Omron Sysmac Studio project INV00x_MX2_ECT (Sysmac Studio 1.45.1.64010, LibraryProject)
(* Functionblocks that can be used for controlling 3G3MX2 with Omron NJ controller over EtherCAT communication. *)

# Controller new_Controller_0: NX102-9000 version 1.40
Task PrimaryTask (priority 4, period or condition 1000): DEMO_INV012_MX2_Analog_inputs, DEMO_INV000_MX2_Alarm, DEMO_INV001_MX2_ECT, DEMO_INV002_MX2_ECT, DEMO_INV003_MX2_ECT, DEMO_INV010_MX2_ExternalTrip, DEMO_INV011_MX2_Intelligent_inputs

TYPE INV00x_MX2\uWORD_BOOL_MX2 : UNION
    bit : ARRAY[0..15] OF BOOL;
    ch : WORD;
END_UNION END_TYPE
TYPE INV00x_MX2\uBYTE_BOOL_MX2 : UNION
    bit : ARRAY[0..7] OF BOOL;
    value : BYTE;
END_UNION END_TYPE

PROGRAM DEMO_INV000_MX2_Alarm
VAR
    sFB_Activate : BOOL;
    MX2 : INV001_MX2_ECT;
    sFrequence : REAL;
    sFwd : BOOL;
    sRev : BOOL;
    sFault_Reset : BOOL;
    sDuring_FDW : BOOL;
    sDuring_Rev : BOOL;
    sWarning : BOOL;
    sRemote : BOOL;
    sFreq_Match : BOOL;
    sConection_Error : BOOL;
    sFB_Activate_2 : BOOL;
    MX2_2 : INV002_MX2_ECT;
    sFault : BOOL;
    sFrequency_in : REAL;
    sFrequency_out : REAL;
    sFB_Activate_3 : BOOL;
    MX2_3 : INV003_MX2_ECT;
    sAcceleration : REAL;
    sDeceleration : REAL;
    MX2_Alarm : INV000_MX2_Alarm;
    sAlarm_Fault : STRING[256];
    sAlarm_Status : STRING[256];
    sAlarm_code : UINT;
    SDO_Obj_W : _sSDO_ACCESS;
END_VAR
VAR RETAIN
    Write_Data : WORD;
END_VAR
VAR
    EtherCAT_Write_External_Trip : EC_CoESDOWrite;
    Node : UINT;
    MX2_ExternalTrip : INV010_MX2_ExternalTrip;
    ExternalTrip : BOOL;
    Read_DI : BOOL;
    TEST : BOOL;
    test2 : WORD;
    s1 : BOOL;
    s2 : BOOL;
    s3 : BOOL;
    s4 : BOOL;
    s5 : BOOL;
    s6 : BOOL;
    s7 : BOOL;
    sRun_Command : BOOL;
    sRotation_Direction : BOOL;
    sExternal_Trip : BOOL;
    MX2_Intelligent_inputs : INV011_MX2_Intelligent_inputs;
    Analog_Input : BOOL;
    MX2_Analog_Inputs : INV012_MX2_Analog_inputs;
    sAnaloge_Value : REAL;
    MX2_Frequency_reference : UINT;
    MX2_Output_frequency_monitor : UINT;
    MX2_F002_1st_Acceleration_Time_1 : UDINT;
    MX2_F003_1st_Deceleration_Time_1 : UDINT;
    MX2_Coil_Data_0 : WORD;
    MX2_Command : WORD;
    MX2_d081_Fault_Monitor_1_Cause : UINT;
    MX2_d081_Fault_Monitor_1_Inverter_Status : UINT;
    MX2_d130_Analog_voltage_input_FV_monitor : UINT;
    MX2_Status : WORD;
END_VAR

(* Section Section1: ladder, written here as Structured Text *)

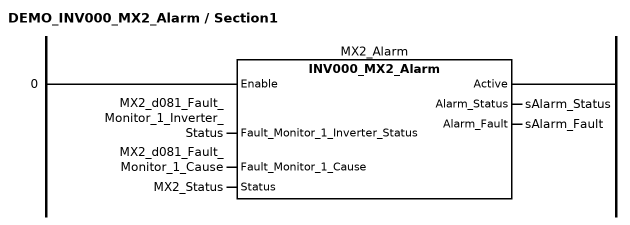
(* Rung 0 *)
MX2_Alarm(Enable := TRUE, Fault_Monitor_1_Inverter_Status := MX2_d081_Fault_Monitor_1_Inverter_Status, Fault_Monitor_1_Cause := MX2_d081_Fault_Monitor_1_Cause, Status := MX2_Status, Alarm_Status => sAlarm_Status, Alarm_Fault => sAlarm_Fault);
END_PROGRAM

PROGRAM DEMO_INV001_MX2_ECT
VAR
    sFB_Activate : BOOL;
    MX2 : INV001_MX2_ECT;
    sFrequence : REAL;
    sFwd : BOOL;
    sRev : BOOL;
    sFault_Reset : BOOL;
    sDuring_FDW : BOOL;
    sDuring_Rev : BOOL;
    sWarning : BOOL;
    sRemote : BOOL;
    sFreq_Match : BOOL;
    sConection_Error : BOOL;
    sFB_Activate_2 : BOOL;
    MX2_2 : INV002_MX2_ECT;
    sFault : BOOL;
    sFrequency_in : REAL;
    sFrequency_out : REAL;
    sFB_Activate_3 : BOOL;
    MX2_3 : INV003_MX2_ECT;
    sAcceleration : REAL;
    sDeceleration : REAL;
    MX2_Alarm : INV000_MX2_Alarm;
    sAlarm_Fault : STRING[256];
    sAlarm_Status : STRING[256];
    sAlarm_code : UINT;
    SDO_Obj_W : _sSDO_ACCESS;
END_VAR
VAR RETAIN
    Write_Data : WORD;
END_VAR
VAR
    EtherCAT_Write_External_Trip : EC_CoESDOWrite;
    Node : UINT;
    MX2_ExternalTrip : INV010_MX2_ExternalTrip;
    ExternalTrip : BOOL;
    Read_DI : BOOL;
    TEST : BOOL;
    test2 : WORD;
    s1 : BOOL;
    s2 : BOOL;
    s3 : BOOL;
    s4 : BOOL;
    s5 : BOOL;
    s6 : BOOL;
    s7 : BOOL;
    sRun_Command : BOOL;
    sRotation_Direction : BOOL;
    sExternal_Trip : BOOL;
    MX2_Intelligent_inputs : INV011_MX2_Intelligent_inputs;
    Analog_Input : BOOL;
    MX2_Analog_Inputs : INV012_MX2_Analog_inputs;
    sAnaloge_Value : REAL;
    MX2_F002_1st_Acceleration_Time_1 : UDINT;
    MX2_F003_1st_Deceleration_Time_1 : UDINT;
    MX2_d081_Fault_Monitor_1_Inverter_Status : UINT;
    MX2_d081_Fault_Monitor_1_Cause : UINT;
    MX2_Coil_Data_0 : WORD;
    MX2_d130_Analog_voltage_input_FV_monitor : UINT;
    sFrequency_0Hz_Warning : BOOL;
    MX2_Frequency_reference : UINT;
    MX2_Output_frequency_monitor : UINT;
    MX2_Command : WORD;
    MX2_Status : WORD;
END_VAR

(* Section Section1: ladder, written here as Structured Text *)

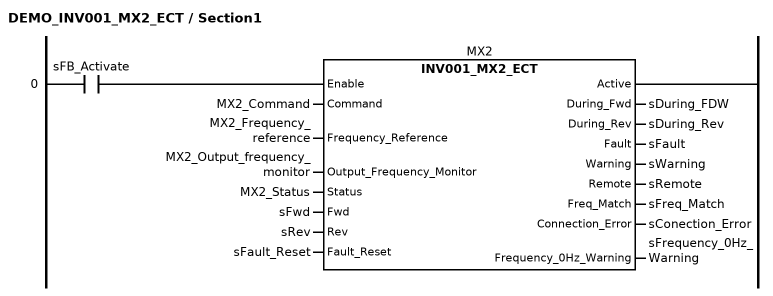
(* Rung 0 *)
MX2(Enable := sFB_Activate, Command := MX2_Command, Frequency_Reference := MX2_Frequency_reference, Output_Frequency_Monitor := MX2_Output_frequency_monitor, Status := MX2_Status, Fwd := sFwd, Rev := sRev, Fault_Reset := sFault_Reset, During_Fwd => sDuring_FDW, During_Rev => sDuring_Rev, Fault => sFault, Warning => sWarning, Remote => sRemote, Freq_Match => sFreq_Match, Connection_Error => sConection_Error, Frequency_0Hz_Warning => sFrequency_0Hz_Warning);
END_PROGRAM

PROGRAM DEMO_INV002_MX2_ECT
VAR
    sFB_Activate : BOOL;
    MX2 : INV001_MX2_ECT;
    sFrequence : REAL;
    sFwd : BOOL;
    sRev : BOOL;
    sFault_Reset : BOOL;
    sDuring_FDW : BOOL;
    sDuring_Rev : BOOL;
    sWarning : BOOL;
    sRemote : BOOL;
    sFreq_Match : BOOL;
    sConection_Error : BOOL;
    sFB_Activate_2 : BOOL;
    MX2_2 : INV002_MX2_ECT;
    sFault : BOOL;
    sFrequency_in : REAL;
    sFrequency_out : REAL;
    sFB_Activate_3 : BOOL;
    MX2_3 : INV003_MX2_ECT;
    sAcceleration : REAL;
    sDeceleration : REAL;
    MX2_Alarm : INV000_MX2_Alarm;
    sAlarm_Fault : STRING[256];
    sAlarm_Status : STRING[256];
    sAlarm_code : UINT;
    SDO_Obj_W : _sSDO_ACCESS;
END_VAR
VAR RETAIN
    Write_Data : WORD;
END_VAR
VAR
    EtherCAT_Write_External_Trip : EC_CoESDOWrite;
    Node : UINT;
    MX2_ExternalTrip : INV010_MX2_ExternalTrip;
    ExternalTrip : BOOL;
    Read_DI : BOOL;
    TEST : BOOL;
    test2 : WORD;
    s1 : BOOL;
    s2 : BOOL;
    s3 : BOOL;
    s4 : BOOL;
    s5 : BOOL;
    s6 : BOOL;
    s7 : BOOL;
    sRun_Command : BOOL;
    sRotation_Direction : BOOL;
    sExternal_Trip : BOOL;
    MX2_Intelligent_inputs : INV011_MX2_Intelligent_inputs;
    Analog_Input : BOOL;
    MX2_Analog_Inputs : INV012_MX2_Analog_inputs;
    sAnaloge_Value : REAL;
    MX2_Command : WORD;
    MX2_Frequency_reference : UINT;
    MX2_Output_frequency_monitor : UINT;
    MX2_Status : WORD;
    MX2_F002_1st_Acceleration_Time_1 : UDINT;
    MX2_F003_1st_Deceleration_Time_1 : UDINT;
    MX2_d081_Fault_Monitor_1_Inverter_Status : UINT;
    MX2_d081_Fault_Monitor_1_Cause : UINT;
    MX2_Coil_Data_0 : WORD;
    MX2_d130_Analog_voltage_input_FV_monitor : UINT;
    sFrequency_0Hz_Warning : BOOL;
END_VAR

(* Section Section1: ladder, written here as Structured Text *)

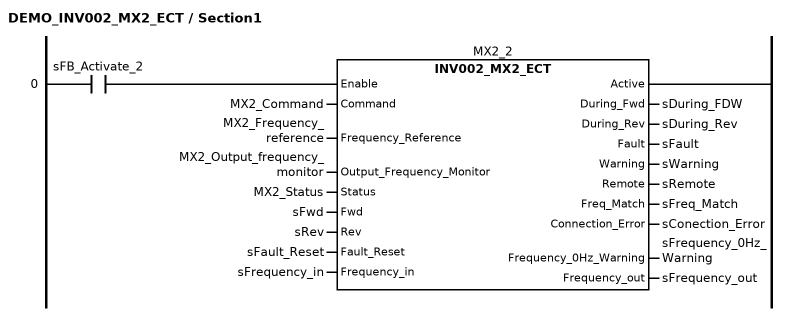
(* Rung 0 *)
MX2_2(Enable := sFB_Activate_2, Command := MX2_Command, Frequency_Reference := MX2_Frequency_reference, Output_Frequency_Monitor := MX2_Output_frequency_monitor, Status := MX2_Status, Fwd := sFwd, Rev := sRev, Fault_Reset := sFault_Reset, Frequency_in := sFrequency_in, During_Fwd => sDuring_FDW, During_Rev => sDuring_Rev, Fault => sFault, Warning => sWarning, Remote => sRemote, Freq_Match => sFreq_Match, Connection_Error => sConection_Error, Frequency_0Hz_Warning => sFrequency_0Hz_Warning, Frequency_out => sFrequency_out);
END_PROGRAM

PROGRAM DEMO_INV003_MX2_ECT
VAR
    sFB_Activate : BOOL;
    MX2 : INV001_MX2_ECT;
    sFrequence : REAL;
    sFwd : BOOL;
    sRev : BOOL;
    sFault_Reset : BOOL;
    sDuring_FDW : BOOL;
    sDuring_Rev : BOOL;
    sWarning : BOOL;
    sRemote : BOOL;
    sFreq_Match : BOOL;
    sConection_Error : BOOL;
    sFB_Activate_2 : BOOL;
    MX2_2 : INV002_MX2_ECT;
    sFault : BOOL;
    sFrequency_in : REAL;
    sFrequency_out : REAL;
    sFB_Activate_3 : BOOL;
    MX2_3 : INV003_MX2_ECT;
    sAcceleration : REAL;
    sDeceleration : REAL;
    MX2_Alarm : INV000_MX2_Alarm;
    sAlarm_Fault : STRING[256];
    sAlarm_Status : STRING[256];
    sAlarm_code : UINT;
    SDO_Obj_W : _sSDO_ACCESS;
END_VAR
VAR RETAIN
    Write_Data : WORD;
END_VAR
VAR
    EtherCAT_Write_External_Trip : EC_CoESDOWrite;
    Node : UINT;
    MX2_ExternalTrip : INV010_MX2_ExternalTrip;
    ExternalTrip : BOOL;
    Read_DI : BOOL;
    TEST : BOOL;
    test2 : WORD;
    s1 : BOOL;
    s2 : BOOL;
    s3 : BOOL;
    s4 : BOOL;
    s5 : BOOL;
    s6 : BOOL;
    s7 : BOOL;
    sRun_Command : BOOL;
    sRotation_Direction : BOOL;
    sExternal_Trip : BOOL;
    MX2_Intelligent_inputs : INV011_MX2_Intelligent_inputs;
    Analog_Input : BOOL;
    MX2_Analog_Inputs : INV012_MX2_Analog_inputs;
    sAnaloge_Value : REAL;
    MX2_Command : WORD;
    MX2_Frequency_reference : UINT;
    MX2_Output_frequency_monitor : UINT;
    MX2_Status : WORD;
    MX2_F002_1st_Acceleration_Time_1 : UDINT;
    MX2_F003_1st_Deceleration_Time_1 : UDINT;
    MX2_d081_Fault_Monitor_1_Inverter_Status : UINT;
    MX2_d081_Fault_Monitor_1_Cause : UINT;
    MX2_Coil_Data_0 : WORD;
    MX2_d130_Analog_voltage_input_FV_monitor : UINT;
    sFrequency_0Hz_Warning : BOOL;
END_VAR

(* Section Section1: ladder, written here as Structured Text *)

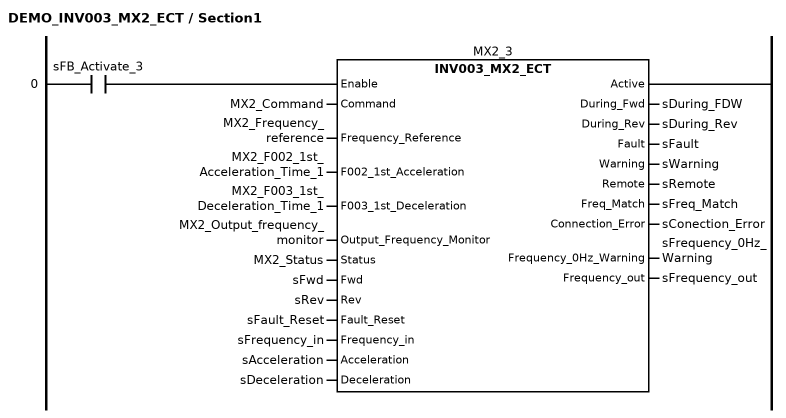
(* Rung 0 *)
MX2_3(Enable := sFB_Activate_3, Command := MX2_Command, Frequency_Reference := MX2_Frequency_reference, F002_1st_Acceleration := MX2_F002_1st_Acceleration_Time_1, F003_1st_Deceleration := MX2_F003_1st_Deceleration_Time_1, Output_Frequency_Monitor := MX2_Output_frequency_monitor, Status := MX2_Status, Fwd := sFwd, Rev := sRev, Fault_Reset := sFault_Reset, Frequency_in := sFrequency_in, Acceleration := sAcceleration, Deceleration := sDeceleration, During_Fwd => sDuring_FDW, During_Rev => sDuring_Rev, Fault => sFault, Warning => sWarning, Remote => sRemote, Freq_Match => sFreq_Match, Connection_Error => sConection_Error, Frequency_0Hz_Warning => sFrequency_0Hz_Warning, Frequency_out => sFrequency_out);
END_PROGRAM

PROGRAM DEMO_INV010_MX2_ExternalTrip
VAR
    sFB_Activate : BOOL;
    MX2 : INV001_MX2_ECT;
    sFrequence : REAL;
    sFwd : BOOL;
    sRev : BOOL;
    sFault_Reset : BOOL;
    sDuring_FDW : BOOL;
    sDuring_Rev : BOOL;
    sWarning : BOOL;
    sRemote : BOOL;
    sFreq_Match : BOOL;
    sConection_Error : BOOL;
    sFB_Activate_2 : BOOL;
    MX2_2 : INV002_MX2_ECT;
    sFault : BOOL;
    sFrequency_in : REAL;
    sFrequency_out : REAL;
    sFB_Activate_3 : BOOL;
    MX2_3 : INV003_MX2_ECT;
    sAcceleration : REAL;
    sDeceleration : REAL;
    MX2_Alarm : INV000_MX2_Alarm;
    sAlarm_Fault : STRING[256];
    sAlarm_Status : STRING[256];
    sAlarm_code : UINT;
    SDO_Obj_W : _sSDO_ACCESS;
END_VAR
VAR RETAIN
    Write_Data : WORD;
END_VAR
VAR
    EtherCAT_Write_External_Trip : EC_CoESDOWrite;
    Node : UINT;
    MX2_ExternalTrip : INV010_MX2_ExternalTrip;
    ExternalTrip : BOOL;
    Read_DI : BOOL;
    TEST : BOOL;
    test2 : WORD;
    s1 : BOOL;
    s2 : BOOL;
    s3 : BOOL;
    s4 : BOOL;
    s5 : BOOL;
    s6 : BOOL;
    s7 : BOOL;
    sRun_Command : BOOL;
    sRotation_Direction : BOOL;
    sExternal_Trip : BOOL;
    MX2_Intelligent_inputs : INV011_MX2_Intelligent_inputs;
    Analog_Input : BOOL;
    MX2_Analog_Inputs : INV012_MX2_Analog_inputs;
    sAnaloge_Value : REAL;
    MX2_Command : WORD;
    MX2_Frequency_reference : UINT;
    MX2_Output_frequency_monitor : UINT;
    MX2_Status : WORD;
    MX2_F002_1st_Acceleration_Time_1 : UDINT;
    MX2_F003_1st_Deceleration_Time_1 : UDINT;
    MX2_d081_Fault_Monitor_1_Inverter_Status : UINT;
    MX2_d081_Fault_Monitor_1_Cause : UINT;
    MX2_Coil_Data_0 : WORD;
    MX2_d130_Analog_voltage_input_FV_monitor : UINT;
END_VAR

(* Section Section1: ladder, written here as Structured Text *)

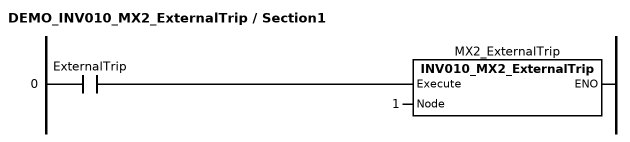
(* Rung 0 *)
MX2_ExternalTrip(Execute := ExternalTrip, Node := 1);
END_PROGRAM

PROGRAM DEMO_INV011_MX2_Intelligent_inputs
VAR
    sFB_Activate : BOOL;
    MX2 : INV001_MX2_ECT;
    sFrequence : REAL;
    sFwd : BOOL;
    sRev : BOOL;
    sFault_Reset : BOOL;
    sDuring_FDW : BOOL;
    sDuring_Rev : BOOL;
    sWarning : BOOL;
    sRemote : BOOL;
    sFreq_Match : BOOL;
    sConection_Error : BOOL;
    sFB_Activate_2 : BOOL;
    MX2_2 : INV002_MX2_ECT;
    sFault : BOOL;
    sFrequency_in : REAL;
    sFrequency_out : REAL;
    sFB_Activate_3 : BOOL;
    MX2_3 : INV003_MX2_ECT;
    sAcceleration : REAL;
    sDeceleration : REAL;
    MX2_Alarm : INV000_MX2_Alarm;
    sAlarm_Fault : STRING[256];
    sAlarm_Status : STRING[256];
    sAlarm_code : UINT;
    SDO_Obj_W : _sSDO_ACCESS;
END_VAR
VAR RETAIN
    Write_Data : WORD;
END_VAR
VAR
    EtherCAT_Write_External_Trip : EC_CoESDOWrite;
    Node : UINT;
    MX2_ExternalTrip : INV010_MX2_ExternalTrip;
    ExternalTrip : BOOL;
    Read_DI : BOOL;
    TEST : BOOL;
    test2 : WORD;
    s1 : BOOL;
    s2 : BOOL;
    s3 : BOOL;
    s4 : BOOL;
    s5 : BOOL;
    s6 : BOOL;
    s7 : BOOL;
    sRun_Command : BOOL;
    sRotation_Direction : BOOL;
    sExternal_Trip : BOOL;
    MX2_Intelligent_inputs : INV011_MX2_Intelligent_inputs;
    Analog_Input : BOOL;
    MX2_Analog_Inputs : INV012_MX2_Analog_inputs;
    sAnaloge_Value : REAL;
    MX2_Command : WORD;
    MX2_Frequency_reference : UINT;
    MX2_Output_frequency_monitor : UINT;
    MX2_Status : WORD;
    MX2_F002_1st_Acceleration_Time_1 : UDINT;
    MX2_F003_1st_Deceleration_Time_1 : UDINT;
    MX2_d081_Fault_Monitor_1_Inverter_Status : UINT;
    MX2_d081_Fault_Monitor_1_Cause : UINT;
    MX2_Coil_Data_0 : WORD;
    MX2_d130_Analog_voltage_input_FV_monitor : UINT;
END_VAR

(* Section Section1: ladder, written here as Structured Text *)

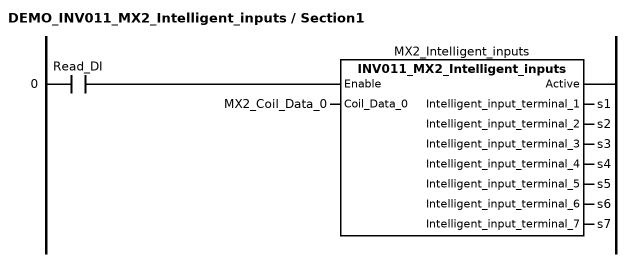
(* Rung 0 *)
MX2_Intelligent_inputs(Enable := Read_DI, Coil_Data_0 := MX2_Coil_Data_0, Intelligent_input_terminal_1 => s1, Intelligent_input_terminal_2 => s2, Intelligent_input_terminal_3 => s3, Intelligent_input_terminal_4 => s4, Intelligent_input_terminal_5 => s5, Intelligent_input_terminal_6 => s6, Intelligent_input_terminal_7 => s7);
END_PROGRAM

PROGRAM DEMO_INV012_MX2_Analog_inputs
VAR
    sFB_Activate : BOOL;
    MX2 : INV001_MX2_ECT;
    sFrequence : REAL;
    sFwd : BOOL;
    sRev : BOOL;
    sFault_Reset : BOOL;
    sDuring_FDW : BOOL;
    sDuring_Rev : BOOL;
    sWarning : BOOL;
    sRemote : BOOL;
    sFreq_Match : BOOL;
    sConection_Error : BOOL;
    sFB_Activate_2 : BOOL;
    MX2_2 : INV002_MX2_ECT;
    sFault : BOOL;
    sFrequency_in : REAL;
    sFrequency_out : REAL;
    sFB_Activate_3 : BOOL;
    MX2_3 : INV003_MX2_ECT;
    sAcceleration : REAL;
    sDeceleration : REAL;
    MX2_Alarm : INV000_MX2_Alarm;
    sAlarm_Fault : STRING[256];
    sAlarm_Status : STRING[256];
    sAlarm_code : UINT;
    SDO_Obj_W : _sSDO_ACCESS;
END_VAR
VAR RETAIN
    Write_Data : WORD;
END_VAR
VAR
    EtherCAT_Write_External_Trip : EC_CoESDOWrite;
    Node : UINT;
    MX2_ExternalTrip : INV010_MX2_ExternalTrip;
    ExternalTrip : BOOL;
    Read_DI : BOOL;
    TEST : BOOL;
    test2 : WORD;
    s1 : BOOL;
    s2 : BOOL;
    s3 : BOOL;
    s4 : BOOL;
    s5 : BOOL;
    s6 : BOOL;
    s7 : BOOL;
    sRun_Command : BOOL;
    sRotation_Direction : BOOL;
    sExternal_Trip : BOOL;
    MX2_Intelligent_inputs : INV011_MX2_Intelligent_inputs;
    Analog_Input : BOOL;
    MX2_Analog_Inputs : INV012_MX2_Analog_inputs;
    sAnaloge_voltage : REAL;
    sAnaloge_current : REAL;
    sAnaloge_voltage_Procentage : REAL;
    sAnaloge_current_Procentage : REAL;
    sAnaloge_voltage_Percentage : REAL;
    sAnaloge_current_Percentage : REAL;
    MX2_Command : WORD;
    MX2_Frequency_reference : UINT;
    MX2_Output_frequency_monitor : UINT;
    MX2_Status : WORD;
    MX2_F002_1st_Acceleration_Time_1 : UDINT;
    MX2_F003_1st_Deceleration_Time_1 : UDINT;
    MX2_d081_Fault_Monitor_1_Inverter_Status : UINT;
    MX2_d081_Fault_Monitor_1_Cause : UINT;
    MX2_Coil_Data_0 : WORD;
    MX2_d130_Analog_voltage_input_FV_monitor : UINT;
    MX2_d131_Analog_current_input_FI_monitor : UINT;
END_VAR

(* Section Section1: ladder, written here as Structured Text *)

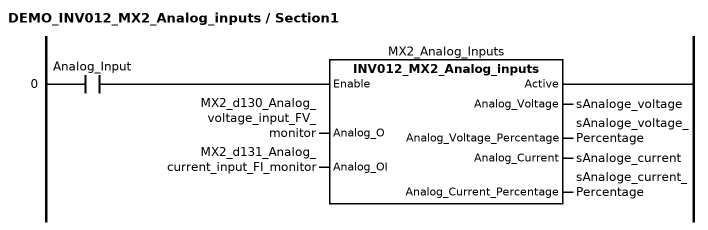
(* Rung 0 *)
MX2_Analog_Inputs(Enable := Analog_Input, Analog_O := MX2_d130_Analog_voltage_input_FV_monitor, Analog_OI := MX2_d131_Analog_current_input_FI_monitor, Analog_Voltage => sAnaloge_voltage, Analog_Voltage_Percentage => sAnaloge_voltage_Percentage, Analog_Current => sAnaloge_current, Analog_Current_Percentage => sAnaloge_current_Percentage);
END_PROGRAM

FUNCTION_BLOCK INV000_MX2_Alarm
(* Alarms from 3G3MX2 *)
VAR
    tmp_Status : INV00x_MX2\uWORD_BOOL_MX2;
END_VAR
VAR_OUTPUT
    Active : BOOL;  (* Functionblock is active *)
    Alarm_Status : STRING[256];
    Alarm_Fault : STRING[256];
END_VAR
VAR_INPUT
    Enable : BOOL;  (* Enables the Functionblock *)
    Fault_Monitor_1_Inverter_Status : UINT;
    Fault_Monitor_1_Cause : UINT;
    Status : WORD;
END_VAR
///FB ON///
Active:=Enable;

///Status extraction///
	tmp_Status.ch := Status;

//If MX2 has an fault the latest fault will be outputted//
IF tmp_Status.bit[3]=TRUE THEN
	
//MX2 Inverter fault factor list name//
CASE Fault_Monitor_1_Cause OF
	00 : 
		Alarm_Fault:='No trip factor';	
	01 : 
		Alarm_Fault:='Overcurrent protection during constant speed';
   	02 : 
		Alarm_Fault:='Overcurrent protection during deceleration';
	03 : 
		Alarm_Fault:='Overcurrent protection during acceleration';
	04 : 
		Alarm_Fault:='Overcurrent protection during stop';
	05 : 
		Alarm_Fault:='Overload protection';
	06 : 
		Alarm_Fault:='Braking resistor overload protection';
	07 : 
		Alarm_Fault:='Overvoltage protection';
	08 : 
		Alarm_Fault:='EEPROM error';
	09 : 
		Alarm_Fault:='Undervoltage protection';
	10 : 
		Alarm_Fault:='Current detector error';
	11 : 
		Alarm_Fault:='CPU error';
	12 : 
		Alarm_Fault:='External trip';
	13 : 
		Alarm_Fault:='USP error';
	14 : 
		Alarm_Fault:='Grounding protection';
	15 : 
		Alarm_Fault:='Incoming overvoltage protection';
	21 : 
		Alarm_Fault:='Abnormal temperature';
	25 : 
		Alarm_Fault:='Main circuit error';
	30 : 
		Alarm_Fault:='Driver error';
	35 : 
		Alarm_Fault:='Thermistor error';
	36 : 
		Alarm_Fault:='Brake error';
	37 : 
		Alarm_Fault:='Emergency shutoff';
	38 : 
		Alarm_Fault:='Overload protection in a low speed range';
	40 : 
		Alarm_Fault:='Digital operator connection error';
	41 : 
		Alarm_Fault:='Modbus communication (Modbus-RTU) error';
	43..45 : 
		Alarm_Fault:='Internal data error';
	50..69 : 
		Alarm_Fault:='Internal data error';	
	80 : 
		Alarm_Fault:='Encoder disconnection';
	81 : 
		Alarm_Fault:='Overspeed';
	83 : 
		Alarm_Fault:='Position control range trip';
	

		
END_CASE;

//MX2 Inverter status at fault occur//


	CASE Fault_Monitor_1_Inverter_Status OF
    	0 : 
			Alarm_Status:='During reset';
		1 : 
			Alarm_Status:='During stop';
		2 : 
			Alarm_Status:='During deceleration';
		3 : 
			Alarm_Status:='At a constant speed';
		4 : 
			Alarm_Status:='During acceleration';
		5 : 
			Alarm_Status:='Operates at frequency = 0';
		6 : 
			Alarm_Status:='During startup';
		7 : 
			Alarm_Status:='DB active (DC injection braking active)';
		8 : 
			Alarm_Status:='During overload limit';
		
	END_CASE;
ELSE
	Alarm_Fault:='No trip factor';	
	Alarm_Status:='--';
	
END_IF;
END_FUNCTION_BLOCK

FUNCTION_BLOCK INV001_MX2_ECT
(* MX2 standard FB *)
VAR
    tmp_freq_in_real : REAL;
    tmp_freq_in_int : UINT;
    tmp_freq_out_real : REAL;
    tmp_freq_out_int : UINT;
    tmp_Command : INV00x_MX2\uWORD_BOOL_MX2;
    tmp_Status : INV00x_MX2\uWORD_BOOL_MX2;
END_VAR
VAR_IN_OUT
    Command : WORD;  (* Inverter Command word *)
    Frequency_Reference : UINT;  (* Specify the frequency in increments of 0.01 Hz *)
    Output_Frequency_Monitor : UINT;  (* Displays the output frequency in increments of 0.01 Hz *)
    Status : WORD;  (* Inverter Status word *)
END_VAR
VAR_OUTPUT
    Active : BOOL;  (* Functionblock is active *)
    During_Fwd : BOOL;  (* 0: Stopped/ during reverse operation 1: During forward operation *)
    During_Rev : BOOL;  (* 0: Stopped/ during forward operation 1: During reverse operation *)
    Fault : BOOL;  (* 0: No error or trip onccurred for the unit 1: Error or trip has occurred for the he unit *)
    Warning : BOOL;  (* 0: No waring onccurred for the unit 1: Warining occurred for the unit *)
    Remote : BOOL;  (* 0: Local (Operations from EtherCAT are disabled) 1: Remote (Operations from EtherCAT are enabled) *)
    Freq_Match : BOOL;  (* 0: During acceleration/deceleration 1: Frequency matched *)
    Connection_Error : BOOL;  (* Connection error between the Optional Unit and inverter *)
    Frequency_0Hz_Warning : BOOL;
END_VAR
VAR_INPUT
    Enable : BOOL;  (* Enables the Functionblock	Enable the Functionblock *)
    Fwd : BOOL;  (* 0: Stop, 1: Forward command *)
    Rev : BOOL;  (* 0: Stop, 1: Reverse command *)
    Fault_Reset : BOOL;  (* Resets an error or trip for the unit *)
END_VAR
///Status extraction///
	tmp_Status.ch := Status;
	During_Fwd := tmp_Status.bit[0];
	During_Rev := tmp_Status.bit[1];
	Fault := tmp_Status.bit[3];
	Warning := tmp_Status.bit[7];
	Remote := tmp_Status.bit[9];
	Freq_Match := tmp_Status.bit[12];
	Connection_Error := tmp_Status.bit[15];

///Command extraction///
IF Enable and Frequency_Reference>1 THEN;
	tmp_Command.bit[0] := Fwd;
	tmp_Command.bit[1] := Rev;
	Active:=TRUE;
ELSE
	tmp_Command.bit[0] := FALSE;
	tmp_Command.bit[1] := FALSE;
	Active:=FALSE;
END_IF;
	tmp_Command.bit[7] := Fault_Reset;
	Command := tmp_Command.ch;

//0 Frequence //
IF Enable and Frequency_Reference>0 and (Fwd or Rev) THEN;
	Frequency_0Hz_Warning:=TRUE;
ELSE
	Frequency_0Hz_Warning:=FALSE;
END_IF;
END_FUNCTION_BLOCK

FUNCTION_BLOCK INV002_MX2_ECT
(* MX2 standard FB & REAL value SP & PV *)
VAR
    tmp_freq_in_real : REAL;
    tmp_freq_in_int : UINT;
    tmp_freq_out_real : REAL;
    tmp_freq_out_int : UINT;
    tmp_Command : INV00x_MX2\uWORD_BOOL_MX2;
    tmp_Status : INV00x_MX2\uWORD_BOOL_MX2;
END_VAR
VAR_IN_OUT
    Command : WORD;  (* Inverter Command word *)
    Frequency_Reference : UINT;  (* Specify the frequency in increments of 0.01 Hz *)
END_VAR
VAR_INPUT
    Output_Frequency_Monitor : UINT;  (* Displays the output frequency in increments of 0.01 Hz *)
END_VAR
VAR_IN_OUT
    Status : WORD;  (* Inverter Status word *)
END_VAR
VAR_OUTPUT
    Active : BOOL;  (* Functionblock is active *)
    During_Fwd : BOOL;  (* 0: Stopped/ during reverse operation 1: During forward operation *)
    During_Rev : BOOL;  (* 0: Stopped/ during forward operation 1: During reverse operation *)
    Fault : BOOL;  (* 0: No error or trip onccurred for the unit 1: Error or trip has occurred for the he unit *)
    Warning : BOOL;  (* 0: No waring onccurred for the unit 1: Warining occurred for the unit *)
    Remote : BOOL;  (* 0: Local (Operations from EtherCAT are disabled) 1: Remote (Operations from EtherCAT are enabled) *)
    Freq_Match : BOOL;  (* 0: During acceleration/deceleration 1: Frequency matched *)
    Connection_Error : BOOL;  (* Connection error between the Optional Unit and inverter *)
    Frequency_0Hz_Warning : BOOL;
END_VAR
VAR_INPUT
    Enable : BOOL;  (* Enables the Functionblock	Enable the Functionblock *)
    Fwd : BOOL;  (* 0: Stop, 1: Forward command *)
    Rev : BOOL;  (* 0: Stop, 1: Reverse command *)
    Fault_Reset : BOOL;  (* Resets an error or trip for the unit *)
    Frequency_in : REAL;  (* Specify the set point frequency in 0.01 Hz *)
END_VAR
VAR_OUTPUT
    Frequency_out : REAL;  (* Shows the frequency in 0.01 Hz *)
END_VAR
///Status extraction///
	tmp_Status.ch := Status;
	During_Fwd := tmp_Status.bit[0];
	During_Rev := tmp_Status.bit[1];
	Fault := tmp_Status.bit[3];
	Warning := tmp_Status.bit[7];
	Remote := tmp_Status.bit[9];
	Freq_Match := tmp_Status.bit[12];
	Connection_Error := tmp_Status.bit[15];

///Command extraction///
IF Enable And Frequency_in>0.01 THEN; 
	tmp_Command.bit[0] := Fwd;
	tmp_Command.bit[1] := Rev;
	Active:=TRUE;
ELSE
	tmp_Command.bit[0] := FALSE;
	tmp_Command.bit[1] := FALSE;
	Active:=FALSE;
END_IF;
	tmp_Command.bit[7] := Fault_Reset;
	Command := tmp_Command.ch;

///Frequence form a REAL value///
IF Frequency_in>0.01 THEN;
	tmp_freq_in_real:=Frequency_in*100;
	tmp_freq_in_int:=REAL_TO_UINT(tmp_freq_in_real);
	Frequency_Reference:=tmp_freq_in_int;
END_IF;

//Convert Output_Frequency_Monitor to a REAL value//
	tmp_freq_out_int:=Output_Frequency_Monitor;
	tmp_freq_out_real:=UINT_TO_REAL(tmp_freq_out_int);
	Frequency_out:=tmp_freq_out_real/100.0;
	
//0 Frequence //
IF Enable and Frequency_in>0.01 and (Fwd or Rev) THEN;
	Frequency_0Hz_Warning:=TRUE;
ELSE
	Frequency_0Hz_Warning:=FALSE;
END_IF;
END_FUNCTION_BLOCK

FUNCTION_BLOCK INV003_MX2_ECT
(* MX2 standard FB & Acceleration/Deceleration Time & REAL value SP & PV *)
VAR
    tmp_freq_in_real : REAL;
    tmp_freq_in_int : UINT;
    tmp_freq_out_real : REAL;
    tmp_freq_out_int : UINT;
    tmp_acc_real : REAL;
    tmp_acc_int : INT;
    tmp_dec_real : REAL;
    tmp_dec_int : INT;
    tmp_Command : INV00x_MX2\uWORD_BOOL_MX2;
    tmp_Status : INV00x_MX2\uWORD_BOOL_MX2;
END_VAR
VAR_IN_OUT
    Command : WORD;  (* Inverter Command word *)
    Frequency_Reference : UINT;  (* Specify the frequency in increments of 0.01 Hz *)
    F002_1st_Acceleration : UDINT;
    F003_1st_Deceleration : UDINT;
END_VAR
VAR_INPUT
    Output_Frequency_Monitor : UINT;  (* Displays the output frequency in increments of 0.01 Hz *)
END_VAR
VAR_IN_OUT
    Status : WORD;  (* Inverter Status word *)
END_VAR
VAR_OUTPUT
    Active : BOOL;  (* Functionblock is active *)
    During_Fwd : BOOL;  (* 0: Stopped/ during reverse operation 1: During forward operation *)
    During_Rev : BOOL;  (* 0: Stopped/ during forward operation 1: During reverse operation *)
    Fault : BOOL;  (* 0: No error or trip onccurred for the unit 1: Error or trip has occurred for the he unit *)
    Warning : BOOL;  (* 0: No waring onccurred for the unit 1: Warining occurred for the unit *)
    Remote : BOOL;  (* 0: Local (Operations from EtherCAT are disabled) 1: Remote (Operations from EtherCAT are enabled) *)
    Freq_Match : BOOL;  (* 0: During acceleration/deceleration 1: Frequency matched *)
    Connection_Error : BOOL;  (* Connection error between the Optional Unit and inverter *)
    Frequency_0Hz_Warning : BOOL;
    Frequency_out : REAL;  (* Shows the frequency in 0.01 Hz *)
END_VAR
VAR_INPUT
    Enable : BOOL;  (* Enables the Functionblock	Enable the Functionblock *)
    Fwd : BOOL;  (* 0: Stop, 1: Forward command *)
    Rev : BOOL;  (* 0: Stop, 1: Reverse command *)
    Fault_Reset : BOOL;  (* Resets an error or trip for the unit *)
    Frequency_in : REAL;  (* Specify the set point frequency in 0.01 Hz *)
    Acceleration : REAL;  (* Specify the Acceleration set point in seconds *)
    Deceleration : REAL;  (* Specify the Acceleration set point in seconds *)
END_VAR
///Status extraction///
	tmp_Status.ch := Status;
	During_Fwd := tmp_Status.bit[0];
	During_Rev := tmp_Status.bit[1];
	Fault := tmp_Status.bit[3];
	Warning := tmp_Status.bit[7];
	Remote := tmp_Status.bit[9];
	Freq_Match := tmp_Status.bit[12];
	Connection_Error := tmp_Status.bit[15];

///Command extraction///
IF Enable and Frequency_in>0.01 THEN;
	tmp_Command.bit[0] := Fwd;
	tmp_Command.bit[1] := Rev;
	Active:=TRUE;
ELSE
	tmp_Command.bit[0] := FALSE;
	tmp_Command.bit[1] := FALSE;
	Active:=FALSE;
END_IF;
	tmp_Command.bit[7] := Fault_Reset;
	Command := tmp_Command.ch;

///Frequence form a REAL value///
IF Frequency_in>0.01 THEN;
	tmp_freq_in_real:=Frequency_in*100;
	tmp_freq_in_int:=REAL_TO_UINT(tmp_freq_in_real);
	Frequency_Reference:=tmp_freq_in_int;
END_IF;

//Convert Output_Frequency_Monitor to a REAL value//
	tmp_freq_out_int:=Output_Frequency_Monitor;
	tmp_freq_out_real:=UINT_TO_REAL(tmp_freq_out_int);
	Frequency_out:=tmp_freq_out_real/100.0;
	
//Acceleration/Deceleration Time  in REAL value//
IF Acceleration>0.01 THEN;
	tmp_acc_real:=Acceleration*100;
	tmp_acc_int:=REAL_TO_INT(tmp_acc_real);
	F002_1st_Acceleration:=tmp_acc_int;
END_IF;

IF Deceleration>0.01 THEN;
	tmp_dec_real:=Deceleration*100;
	tmp_dec_int:=REAL_TO_INT(tmp_dec_real);
	F003_1st_Deceleration:=tmp_dec_int;
END_IF;
	
//0 Frequence //
IF Enable and Frequency_in>0.01 and (Fwd or Rev) THEN;
	Frequency_0Hz_Warning:=TRUE;
ELSE
	Frequency_0Hz_Warning:=FALSE;
END_IF;
END_FUNCTION_BLOCK

FUNCTION_BLOCK INV010_MX2_ExternalTrip
(* MX2 External Trip FB *)
VAR
    EtherCAT_Write_External_Trip : EC_CoESDOWrite;
    SDO_Obj_W : _sSDO_ACCESS;
END_VAR
VAR RETAIN
    Write_ExternalTrip : WORD := 8;
    Reset_ExternalTrip : WORD := 0;
END_VAR
VAR
    EtherCAT_Reset_External_Trip : EC_CoESDOWrite;
END_VAR
VAR_INPUT
    Execute : BOOL;  (* Executes the Functionblock *)
    Node : UINT;
END_VAR
VAR
    _e1 : R_TRIG;
    _e2 : F_TRIG;
END_VAR
(* ladder, written here as Structured Text *)

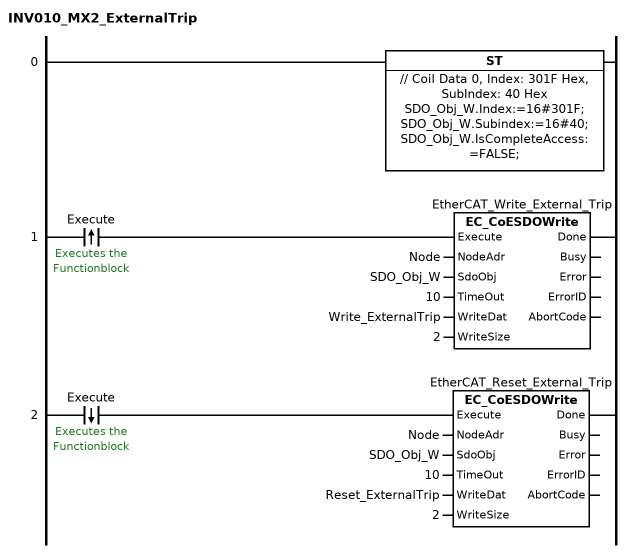
(* Rung 0 *)
// Coil Data 0, Index: 301F Hex, SubIndex: 40 Hex
SDO_Obj_W.Index:=16#301F;
SDO_Obj_W.Subindex:=16#40;
SDO_Obj_W.IsCompleteAccess:=FALSE;
(* Rung 1 *)
_e1(CLK := Execute);
EtherCAT_Write_External_Trip(Execute := _e1.Q, NodeAdr := Node, SdoObj := SDO_Obj_W, TimeOut := 10, WriteDat := Write_ExternalTrip, WriteSize := 2);
(* Rung 2 *)
_e2(CLK := Execute);
EtherCAT_Reset_External_Trip(Execute := _e2.Q, NodeAdr := Node, SdoObj := SDO_Obj_W, TimeOut := 10, WriteDat := Reset_ExternalTrip, WriteSize := 2);
END_FUNCTION_BLOCK

FUNCTION_BLOCK INV011_MX2_Intelligent_inputs
(* MX2 digital Inputs s1-s7 FB *)
VAR
    tmp_Coil_Data_0 : INV00x_MX2\uWORD_BOOL_MX2;
END_VAR
VAR_INPUT
    Enable : BOOL;  (* Enables the Functionblock *)
    Coil_Data_0 : WORD;
END_VAR
VAR_OUTPUT
    Active : BOOL;  (* Functionblock is active *)
    Intelligent_input_terminal_1 : BOOL;  (* 1: ON, 0: OFF *)
    Intelligent_input_terminal_2 : BOOL;  (* 1: ON, 0: OFF *)
    Intelligent_input_terminal_3 : BOOL;  (* 1: ON, 0: OFF *)
    Intelligent_input_terminal_4 : BOOL;  (* 1: ON, 0: OFF *)
    Intelligent_input_terminal_5 : BOOL;  (* 1: ON, 0: OFF *)
    Intelligent_input_terminal_6 : BOOL;  (* 1: ON, 0: OFF *)
    Intelligent_input_terminal_7 : BOOL;  (* 1: ON, 0: OFF *)
END_VAR
// Coil Data 0 to internal uWORD_BOOL_MX2 data type
tmp_Coil_Data_0.ch:=Coil_Data_0;

//Intelligent input terminal (OUT)
IF Enable THEN
Intelligent_input_terminal_1:=tmp_Coil_Data_0.bit[7];
Intelligent_input_terminal_2:=tmp_Coil_Data_0.bit[8];
Intelligent_input_terminal_3:=tmp_Coil_Data_0.bit[9];
Intelligent_input_terminal_4:=tmp_Coil_Data_0.bit[10];
Intelligent_input_terminal_5:=tmp_Coil_Data_0.bit[11];
Intelligent_input_terminal_6:=tmp_Coil_Data_0.bit[12];
Intelligent_input_terminal_7:=tmp_Coil_Data_0.bit[13];
Active:=TRUE;

Else;
Intelligent_input_terminal_1:=FALSE;
Intelligent_input_terminal_2:=FALSE;
Intelligent_input_terminal_3:=FALSE;
Intelligent_input_terminal_4:=FALSE;
Intelligent_input_terminal_5:=FALSE;
Intelligent_input_terminal_6:=FALSE;
Intelligent_input_terminal_7:=FALSE;
Active:=FALSE;

END_IF;
END_FUNCTION_BLOCK

FUNCTION_BLOCK INV012_MX2_Analog_inputs
(* MX2 FB Displays the analog input O or OI value. *)
VAR
    tmp_Analog_Voltage_Bits : REAL;
    tmp_Analog_Current_Bits : REAL;
END_VAR
VAR_INPUT
    Enable : BOOL;  (* Enables the Functionblock *)
    Analog_O : UINT;  (* Analog voltage input FV monitor *)
    Analog_OI : UINT;  (* Analog current input FI monitor *)
END_VAR
VAR_OUTPUT
    Active : BOOL;  (* Functionblock is active *)
    Analog_Voltage : REAL;  (* Voltage in, it displays the inputed value for the terminal FV (0V to 10.9 V) *)
    Analog_Voltage_Percentage : REAL;  (* Voltage In, 0-100% *)
    Analog_Current : REAL;  (* Current in, it displays the inputed value for the terminal FI (4mA to 23.3 mA) *)
    Analog_Current_Percentage : REAL;  (* Current in, 0-100% *)
END_VAR
// move to internal value
	tmp_Analog_Voltage_Bits:=Analog_O;
	tmp_Analog_Current_Bits:=Analog_OI;


IF Enable THEN
//This function is to monitor the value of the analog voltage that is input to the analog voltage reference terminal FV for frequency reference input.//

	Analog_Voltage:=ScaleTrans(SclIn:=tmp_Analog_Voltage_Bits, X0:=0, Y0:=0, X1:=1023, Y1:=10.9);


//This function is to monitor the value of the analog current that is input to the analog voltage reference terminal FI for frequency reference input.//

	Analog_Current:=ScaleTrans(SclIn:=tmp_Analog_Current_Bits, X0:=0, Y0:=4, X1:=1023, Y1:=23.3);

//Percentage of the analog values
//Voltage

	Analog_Voltage_Percentage:=tmp_Analog_Voltage_Bits/1023*100;

//Current

	Analog_Current_Percentage:=tmp_Analog_Current_Bits/1023*100;


Active:=TRUE;

ELSE;
	Analog_Voltage:=0;
	Analog_Current:=0;
	
	Analog_Voltage_Percentage:=0;
	Analog_Current_Percentage:=0;
	
Active:=FALSE;

END_IF;
END_FUNCTION_BLOCK